// TIA Portal V17 export
// export: Created 2024-08-20T10:59:44.5492605Z, ExportSetting WithDefaults, DisplayName Totally Integrated Automation Portal, DisplayVersion V17 Update 4, DisplayName TIA Portal Openness, DisplayVersion V17 Update 4, DisplayName TIA Portal Version Control Interface, DisplayVersion V17, DisplayName STEP 7 Professional, DisplayVersion V17 Update 4, DisplayName STEP 7 Safety, DisplayVersion V17, DisplayName WinCC Advanced, DisplayVersion V17 Update 4
DATA_BLOCK "MODBUS_DB"   // DB102
VERSION : 0.1
// stored: AutoNumber false, DBAccessibleFromOPCUA true, InstanceOfName MODBUS, InstanceOfType FB
"MODBUS"
   // VAR
   //    TEFC0 { S7_SetPoint := 'True'} : TON_TIME;
   //    INI_MOD { S7_SetPoint := 'True'} : TON_TIME;
   //    TEFC1 { S7_SetPoint := 'True'} : TON_TIME;
   //    TEFC2 { S7_SetPoint := 'True'} : TON_TIME;
   //    TEFC3 { S7_SetPoint := 'True'} : TON_TIME;
   //    TEFC4 { S7_SetPoint := 'True'} : TON_TIME;
   //    TEFC5 { S7_SetPoint := 'True'} : TON_TIME;
   //    TEFC6 { S7_SetPoint := 'True'} : TON_TIME;
   //    TEFC7 { S7_SetPoint := 'True'} : TON_TIME;
   //    TEFC8 { S7_SetPoint := 'True'} : TON_TIME;
   //    TEFC9 { S7_SetPoint := 'True'} : TON_TIME;
   //    TEFC10 { S7_SetPoint := 'True'} : TON_TIME;
   //    TEFC11 { S7_SetPoint := 'True'} : TON_TIME;
   //    TEFC12 { S7_SetPoint := 'True'} : TON_TIME;
   //    TEFC13 { S7_SetPoint := 'True'} : TON_TIME;
   //    TEFC14 { S7_SetPoint := 'True'} : TON_TIME;
   //    TEFC15 { S7_SetPoint := 'True'} : TON_TIME;
   //    TEFC16 { S7_SetPoint := 'True'} : TON_TIME;
   //    TEFC17 { S7_SetPoint := 'True'} : TON_TIME;
   //    TEFC18 { S7_SetPoint := 'True'} : TON_TIME;
   //    TEFC19 { S7_SetPoint := 'True'} : TON_TIME;
   //    TEFC20 { S7_SetPoint := 'True'} : TON_TIME;
   //    TEFC21 { S7_SetPoint := 'True'} : TON_TIME;
   //    TEFC22 { S7_SetPoint := 'True'} : TON_TIME;
   //    TEFC23 { S7_SetPoint := 'True'} : TON_TIME;
   //    TEFC24 { S7_SetPoint := 'True'} : TON_TIME;
   //    TEFC25 { S7_SetPoint := 'True'} : TON_TIME;
   //    TEFC26 { S7_SetPoint := 'True'} : TON_TIME;
   //    TEFC27 { S7_SetPoint := 'True'} : TON_TIME;
   //    TEFC28 { S7_SetPoint := 'True'} : TON_TIME;
   // END_VAR
BEGIN
END_DATA_BLOCK
